// TIA Portal V20 export
DATA_BLOCK "HmiInterface"   // DB160
// stored: Access Published, MemoryReserve 100, Namespace Unit1.Em1
   VAR
      em : "LAF_typeEmInterface";
      stacker2NgBox : "LER_typeSequenceInterface";
      cmStacker2NgBoxDetect : "LBC_typeDigitalSignalInterface";
      cmStacker2NgBoxFullDetect : "LBC_typeDigitalSignalInterface";
      cmStacker2NgBoxLoadingUpDown : "LBC_typeTwoWayActuatorInterface";
      cmStacker2NgBoxUnitMoverBwdFwd : "LBC_typeTwoWayActuatorInterface";
      cmStacker2NgBoxClampLeftOpenClose : "LBC_typeTwoWayActuatorInterface";
      cmStacker2NgBoxClampRightOpenClose : "LBC_typeTwoWayActuatorInterface";
      cmStacker2NgBoxClampMoverOpenClose : "LBC_typeTwoWayActuatorInterface";
      cmStacker2NgBoxLiftDownUp : "LBC_typeTwoWayActuatorInterface";
      cmStacker2NgBoxLockDownUp : "LBC_typeTwoWayActuatorInterface";
      intCondition : "Unit1.Em1.typeIntConditionHmiInterface";
   END_VAR
BEGIN
END_DATA_BLOCK
